// TIA Portal V20 export
// export: Created 2026-04-28T10:07:59.5430777Z, ExportSetting WithDefaults, DisplayName Totally Integrated Automation Portal, DisplayVersion V20, DisplayName TIA Portal Openness, DisplayVersion V20, DisplayName TIA Portal Version Control Interface, DisplayVersion V20, DisplayName SINAMICS Startdrive Advanced, DisplayVersion V20, DisplayName SINAMICS Startdrive G130, G150, S120, S150, SINAMICS MV, G220, S200, S210, DisplayVersion V20, DisplayName SINAMICS Startdrive G110M, G120, G120C, G120D, G120P, G115D, DisplayVersion V20, DisplayName STEP 7 Professional, DisplayVersion V20, DisplayName STEP 7 Safety, DisplayVersion V20, DisplayName WinCC Basic/Comfort/Advanced, DisplayVersion V20, DisplayName WinCC Unified, DisplayVersion V20
TYPE "Daten_SPT_20"
// stored: IsFailsafeCompliant false
   STRUCT
      xTower : Bool := false;   // Selection Tower
      xSpDrTe : Bool := false;   // Selection Spray draying plant temperature 1
      iTakt_1_SpT : DInt := 0;   // Interval for recording the measured values
      iAnzWerte_1_SpT : DInt := 0;   // Number of measured values
      xSpDrTe2 : Bool := false;   // Selection Spray draying plant temperature 2
      iTakt_2_SpT : DInt := 0;   // Interval for recording the measured values
      iAnzWerte_2_SpT : DInt := 0;   // Number of measured values
      xSpDrTe3 : Bool := false;   // Selection Spray draying plant temperature 3
      iTakt_3_SpT : DInt := 0;   // Interval for recording the measured values
      iAnzWerte_3_SpT : DInt := 0;   // Number of measured values
      xSpDrTe4 : Bool := false;   // Selection Spray draying plant temperature 4
      iTakt_4_SpT : DInt := 0;   // Interval for recording the measured values
      iAnzWerte_4_SpT : DInt := 0;   // Number of measured values
      xPrTo : Bool := false;   // Selection negative pressure tower
      RangePrTo : DInt := 0;   // Measuring range negative pressure tower
      txt_rPrToMa : DInt := 0;   // Pressure in tower Limit
      txt_max_rPrToMa : DInt := 0;   // Pressure in tower max.
      iTakt_PrTo : DInt := 0;   // Interval for recording the measured values
      iAnzWerte_PrTo : DInt := 0;   // Number of measured values
      xKnVa_Gr1 : Bool := false;   // Selection of knock valves group 1
      t_iKnValve_Gr1 : Time := T#0MS;   // Knock valves group 1 switch-on time
      t_iKnBreake_Gr1 : Time := T#0MS;   // Knock valves group 1 pause time
      xKnVa_Gr2 : Bool := false;   // Selection of knock valves group 2
      t_iKnValve_Gr2 : Time := T#0MS;   // Knock valves group 2 switch-on time
      t_iKnBreake_Gr2 : Time := T#0MS;   // Knock valves group 2 pause time
      xCamera : Bool := false;   // Selection camera
      xPress24_4mA : Bool := false;   // Signal 20-4 mA
      xCleanDoor : Bool := false;   // Selection cleaning door monitoring
      xOptKnVa : Bool := false;   // Selection of knocker valves automatically
      xCleanDev_Ext : Bool;   // Option: External cleaning unit
      i_rExAiTe : DInt;   // Exhaust air Temperature Cleaning
      i_rHoAiTe : DInt;   // Hot air temperature Cleaning
      xPrTo_Sensor2 : Bool := false;   // Selection of negative pressure sensors from -100 to 100 mBar Sensor type 2 = 1
      xPrToCtrl_Intervall : Bool := false;   // Selection Negative pressure tower monitoring at defined intervals
      txt_rPrToCtrl_Up : DInt := 0;   // Selection Negative pressure tower monitoring at defined intervals Up
      txt_rPrToCtrl_Down : DInt := 0;   // Selection Negative pressure tower monitoring at defined intervals Below
      RangePrTo_D20 : DInt := 0;   // Measuring range negative pressure tower
      txt_rPrToMa_D20 : DInt := 0;   // Pressure in tower Limit
      txt_max_rPrToMa_D20 : DInt := 0;   // Pressure in tower max.
   END_STRUCT;
END_TYPE
